// LS Electric XG5000 project: 동남142
// PLC NewPLC
// module base 0 slot 0: 입출력 모듈:XBC-DN/DP14E (DC 24V 입력 8점, 트랜지스터 출력 6점)

PROGRAM NewProgram (task: 스캔 프로그램)

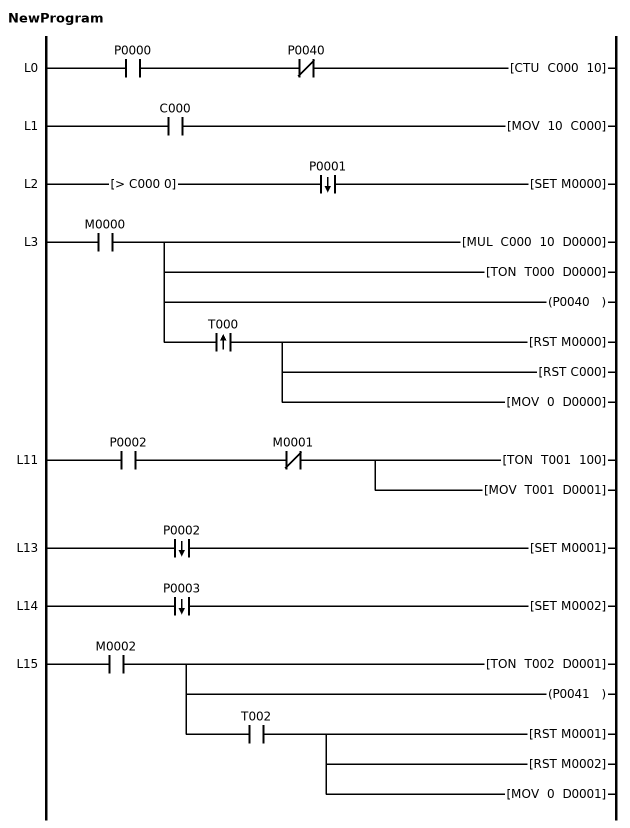
; L0
LOAD      P0000
AND NOT   P0040
CTU       C000 10
; L1
LOAD      C000
MOV       10 C000
; L2
LOAD>     C000 0
ANDN      P0001
SET       M0000
; L3
LOAD      M0000
MUL       C000 10 D0000
TON       T000 D0000
OUT       P0040
ANDP      T000
RST       M0000
RST       C000
MOV       0 D0000
; L11
LOAD      P0002
AND NOT   M0001
TON       T001 100
MOV       T001 D0001
; L13
LOADN     P0002
SET       M0001
; L14
LOADN     P0003
SET       M0002
; L15
LOAD      M0002
TON       T002 D0001
OUT       P0041
AND       T002
RST       M0001
RST       M0002
MOV       0 D0001